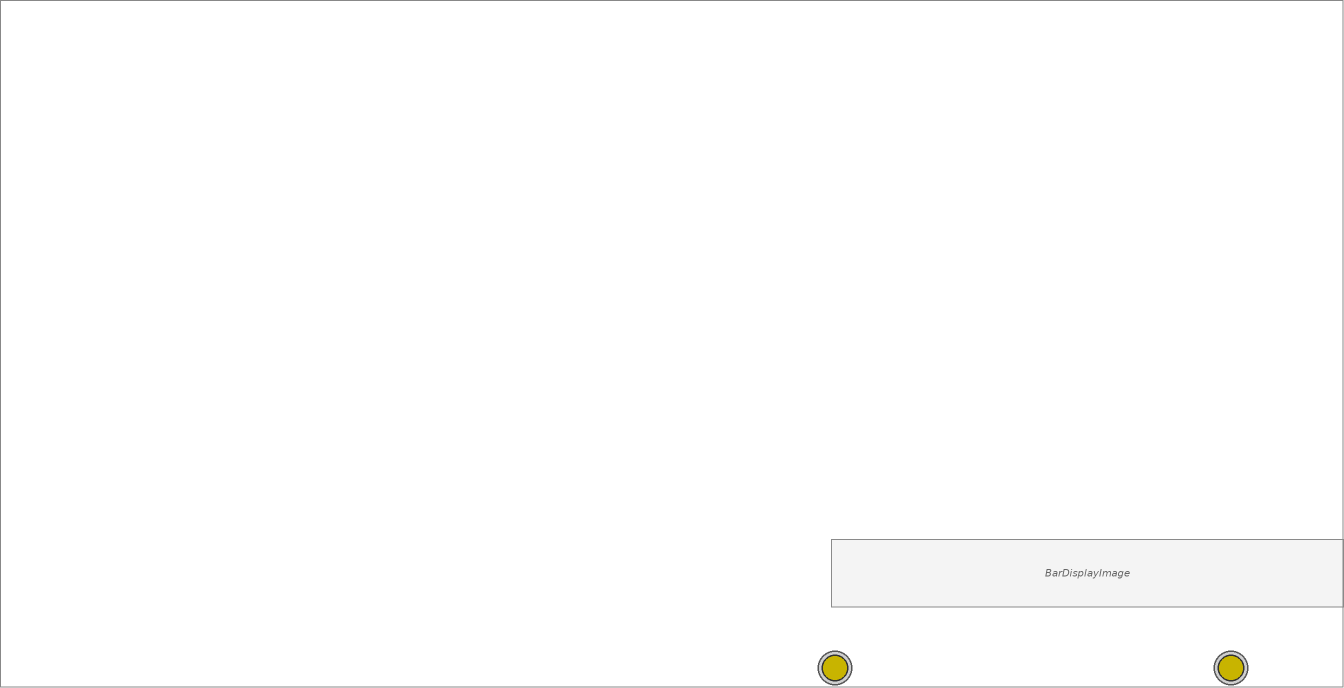
VISUALIZATION Visualization  // 1344x688
    BarDisplayImage (831,539 513x68), style: BarDisplayImage-Gray, scale format: %.1f, scale 0..100
    Lamp1 (815,648 40x40), style: Lamp-Lamp1-Yellow
    Lamp1 (1211,648 40x40), style: Lamp-Lamp1-Yellow
END_VISUALIZATION

(* stored: Version 1.1.0.1
   Visu Visualization: Id {acdf6df7-f660-43ea-9959-7848ba75593b} *)
